INTERFACE Callback

// This is method get's exectued by the framework when the callback is triggered.
// It returns a step number which might be used together with Await to jump to a certain chain step
// after the callback code has been executed.
METHOD execute : UDINT
VAR_INPUT
END_VAR
END_METHOD

END_INTERFACE

(* stored: Version 1.1.0.1, ProductVersion 3.1.4024.12
   Itf Callback: Id {7a36e852-63f5-4890-a3a7-b5281ee647d7}
   Method execute: Id {c9344fd3-d588-4c0d-bd17-31969dad6844} *)
